# EPICS autosave request: iocBoot/iocTimRx/auto_settings.req
file "TimRx_settings.req",                P=$(P),  R=$(R)
